INTERFACE ICylinder

METHOD M_StateMachine : BOOL
VAR_INPUT
	bPosLeftReq  : BOOL;
	bPosRightReq : BOOL;
END_VAR
VAR_OUTPUT
	bAtLeftPos   : BOOL;
	bAtRightPos  : BOOL; 
END_VAR
END_METHOD

PROPERTY P_TimerValue : LREAL
GET
END_GET
SET
END_SET
END_PROPERTY

END_INTERFACE

(* stored: Version 1.1.0.1, ProductVersion 3.1.4024.11
   Itf ICylinder: Id {a72b46da-34d1-4f4e-912c-cc665256fc13}
   Method M_StateMachine: Id {b552e9f9-2368-4f99-80cb-39874c0d68b3}
   Property P_TimerValue: Id {5bdd60c0-9652-4432-89e3-97ab36cfddec}
   Get Get: Id {03f752bf-61e0-4186-ba52-58c2e1a3be7b}
   Set Set: Id {acb36025-fc73-4b83-ae12-5f802808cf8f} *)
